(* CODESYS project lclsmotioncontrol.library
   Company: SLAC
   Title: LCLS Motion Control
   Description: A library containing general use motion control POUs for LCLS.
   Placeholder: LCLS Motion Control
   Author: Alex Wallace
   Version: 0.1.2

Project tree, tasks and I/O mapping:
  libraries: LCLS General, * (SLAC); Tc2_MC2, * (Beckhoff Automation GmbH); Tc2_Standard, * (Beckhoff Automation GmbH); Tc2_System, * (Beckhoff Automation GmbH); Tc2_Utilities, * (Beckhoff Automation GmbH); VisuDialogs, * (System)
  POUs/
    GeneralMotion/
      data type E_AxisMotionState
      data type E_AxisMoveMode
      function block FB_BasicAxisControl [ST]: ActError, ActMove, ActPower
      data type ST_BasicAxis
  Version/
    global variables Global_Version
  VISUs/
    visualisation Basic_Axis_PTP
  visualisation Basic_Axis_PTP
  image pool MotionImagePool
  00000000-0000-0000-0000-000000000000|HMI_Images\ccw-icon.svg
  00000000-0000-0000-0000-000000000000|HMI_Images\abs-go-icon.svg
  00000000-0000-0000-0000-000000000000|HMI_Images\rel-cc-icon.svg
  00000000-0000-0000-0000-000000000000|HMI_Images\rel-plus-icon.svg
  00000000-0000-0000-0000-000000000000|HMI_Images\rel-minus-icon.svg
  00000000-0000-0000-0000-000000000000|HMI_Images\stop-icon.svg
*)

// POUs/GeneralMotion/E_AxisMotionState
TYPE E_AxisMotionState :
(
	Init := 10,
	MoveEnabled := 3000,
	Error := 9000
);
END_TYPE

// POUs/GeneralMotion/E_AxisMoveMode
TYPE E_AxisMoveMode :
(
	Hold := 0,
	MoveAbs	:= 1,
	MoveRel	:= 2
) WORD;
END_TYPE

// POUs/GeneralMotion/ST_BasicAxis
TYPE ST_BasicAxis :
STRUCT

(* Controls *)
xEnable	:	BOOL;
rReqAbsPos	:	LREAL;
rReqRelPos	:	LREAL;
xStartRelMovePlus	:	BOOL;
xStartRelMoveMinus	:	BOOL;
xStartAbsMove	:	BOOL;
xStop	:	BOOL;
wMode	:	E_AxisMoveMode;
xReset	:	BOOL;
i_xMotorInterlock	:	BOOL := FALSE; //External motor interlock, overrides axis enable
	
(* Axis motor *)
stAxis	:	AXIS_REF;
lrVelocity	:	LREAL	:=1; //mm/s

eState	:	E_AxisMotionState;

xHiLS	AT %I* :	BOOL;
xLoLS	AT %I* :	BOOL;

END_STRUCT
END_TYPE

// Version/Global_Version
{attribute 'TcGenerated'}
// This function has been automatically generated from the project information.
VAR_GLOBAL CONSTANT
	{attribute 'const_non_replaced'}
	{attribute 'linkalways'}
	stLibVersion_LCLS_Motion_Control : ST_LibVersion := (iMajor := 0, iMinor := 1, iBuild := 2, iRevision := 0, sVersion := '0.1.2');
END_VAR

// POUs/GeneralMotion/FB_BasicAxisControl
FUNCTION_BLOCK FB_BasicAxisControl
VAR_INPUT
END_VAR
VAR_OUTPUT
	q_asResult: ARRAY [1..20] OF STRING;
	q_xError	:	BOOL;
	q_MoveDone	:	BOOL;
END_VAR
VAR_IN_OUT
	iq_Axis	:	ST_BasicAxis;
END_VAR
VAR
	

	mcPower	:	MC_Power;
	mcReset	:	MC_Reset;
	mcMoveAbsolute : MC_MoveAbsolute;
	mcMoveRelative : MC_MoveRelative;
	mcHalt	:	MC_Halt;
	
	//Error Stuff
	indexResult: FB_Index := (LowerLimit:= 1, UpperLimit:=20);
	fbFormatString	:	FB_FormatString;
	
	imcBlockIndex: INT;
	imcBlockIndexPrev : INT;
	
	rtEnable : R_TRIG;
	ftEnable : F_TRIG;
	rtStop	:	R_TRIG;
	rtStartAbsMove	:	R_TRIG;
	rtStartRelMove	:	R_TRIG;
	rReqAbsPosOld: REAL := 0;
	Direction: LREAL := 1;
	i_xMotorInterlock: INT;
	
END_VAR

(* Basic Axis Controls
Alex Wallace, 2016-8-8 

This FB provides limit switch monitoring, and a basic state machine for absolute and relative moves.

We needed a basic control block that would give us some of the functionality of the system manager screen
that is used for commissioning axes.

*)


rtEnable(CLK:=iq_Axis.xEnable);

//Update status
iq_Axis.stAxis();

//Motor Interlock
////////////////////////////////////////////
//If we attempt to enable the motor, but there is an interlock preventing us, log it
IF rtEnable.Q AND NOT iq_Axis.i_xMotorInterlock THEN
	q_asResult[indexResult.IncVal()] := 'Axis enable failed, motor interlock is not satisfied';
END_IF

iq_Axis.xEnable R= NOT iq_Axis.i_xMotorInterlock;
mcPower.Enable := iq_Axis.xEnable AND iq_Axis.i_xMotorInterlock;

ftEnable(CLK:=iq_Axis.xEnable);
//Reset the axis if it is "turned off"/ disabled
IF ftEnable.Q THEN iq_Axis.eState := Init; END_IF

CASE iq_Axis.eState OF
	0: iq_Axis.eState := Init;
	Init:
		(* Start by initializing the motor axis *)
		IF mcPower.Status AND NOT ftEnable.Q THEN //success
			q_asResult[indexResult.IncVal()] := 'Motor init success';
			iq_Axis.eState := MoveEnabled;
		ELSIF mcPower.Error THEN
			mcPower.Enable := FALSE;
			fbFormatString.sFormat:='Init mcPower Error: %#X';
			fbFormatString.arg1:=F_UDINT(mcPower.ErrorID);
			ActError();
		END_IF
		
	MoveEnabled:
		//MoveAbs
		///////////////////////////////////////////////////////
			mcMoveAbsolute.Execute S= iq_Axis.xStartAbsMove AND NOT mcMoveRelative.Busy;
			mcMoveAbsolute.Position := iq_Axis.rReqAbsPos;
			IF mcMoveAbsolute.Done OR 
				mcMoveAbsolute.CommandAborted OR 
				mcMoveAbsolute.Busy THEN
				mcMoveAbsolute.Execute := FALSE;
			ELSIF mcMoveAbsolute.Error THEN
				mcMoveAbsolute.Execute := FALSE;
				fbFormatString.sFormat:='MoveAbsoluteError: %#X'; 
				fbFormatString.arg1:=F_UDINT(mcMoveAbsolute.ErrorID);
				ActError();
			END_IF
		//MoveRel
		//////////////////////////////////////////////////////////////////
			mcMoveRelative.Execute S= (iq_Axis.xStartRelMovePlus OR iq_Axis.xStartRelMoveMinus) AND NOT mcMoveAbsolute.Busy;
			IF iq_Axis.xStartRelMoveMinus THEN Direction := -1; ELSE Direction := 1; END_IF
			mcMoveRelative.Distance := Direction * iq_Axis.rReqRelPos;
			IF mcMoveRelative.Done OR 
				mcMoveRelative.CommandAborted OR 
				mcMoveRelative.Busy THEN 
				mcMoveRelative.Execute := FALSE;
			ELSIF mcMoveRelative.Error THEN
				mcMoveRelative.Execute := FALSE;
				fbFormatString.sFormat:='MoveRelativeError: %#X'; 
				fbFormatString.arg1:=F_UDINT(mcMoveRelative.ErrorID);
				ActError();
			END_IF

		iq_Axis.xStartAbsMove := FALSE;
		iq_Axis.xStartRelMovePlus := FALSE;
		iq_Axis.xStartRelMoveMinus := FALSE;
		//Halt
		mcMoveAbsolute.Execute R= iq_Axis.xStop;
		mcMoveRelative.Execute R= iq_Axis.xStop;
		mcHalt.Execute S= iq_Axis.xStop;
		mcHalt.Execute R= mcHalt.Busy;
		

	Error:
		IF mcReset.Done THEN
			q_xError := FALSE;
			iq_Axis.eState:=Init;
		END_IF
	
END_CASE

//Move done output logic
//Dones aren't reset until the logic block runs again
q_MoveDone := mcMoveRelative.Done OR mcMoveAbsolute.Done;

(* Run the mc blocks *)
ActPower();
iq_Axis.xReset R= mcReset.Done;
mcReset.Execute := iq_Axis.xReset;
mcReset(Axis:=iq_Axis.stAxis);

mcHalt(Axis:=iq_Axis.stAxis);
ActMove();

ACTION ActError:
(* Error action
*)

//Reset the debugging index
iq_Axis.eState := Error;
q_xError	:=	TRUE;
fbFormatString(sOut=>q_asResult[indexResult.IncVal()]);
END_ACTION

ACTION ActMove:
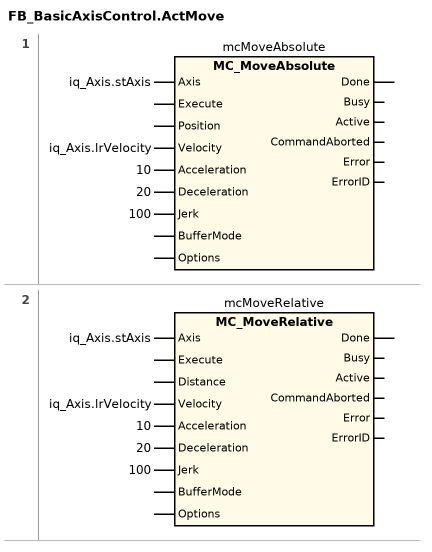
// NETWORK 1
mcMoveAbsolute(
    Axis := iq_Axis.stAxis,
    Velocity := iq_Axis.lrVelocity,
    Acceleration := 10,
    Deceleration := 20,
    Jerk := 100); // MC_MoveAbsolute

// NETWORK 2
mcMoveRelative(
    Axis := iq_Axis.stAxis,
    Velocity := iq_Axis.lrVelocity,
    Acceleration := 10,
    Deceleration := 20,
    Jerk := 100); // MC_MoveRelative
END_ACTION

ACTION ActPower:
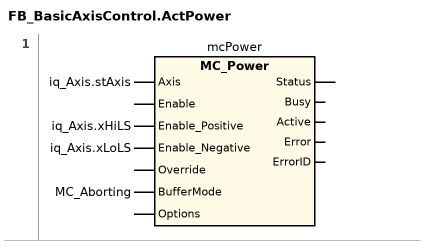
// NETWORK 1
mcPower(
    Axis := iq_Axis.stAxis,
    Enable_Positive := iq_Axis.xHiLS,
    Enable_Negative := iq_Axis.xLoLS,
    BufferMode := MC_Aborting); // MC_Power
END_ACTION

END_FUNCTION_BLOCK

// VISUs/Basic_Axis_PTP
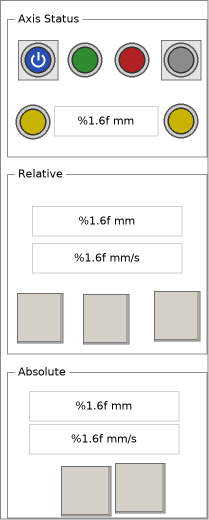
VISUALIZATION Basic_Axis_PTP  // 209x520
VAR_IN_OUT
	stBasicAxis	:	ST_BasicAxis;
END_VAR
    GroupBox (7,11 200x146), "Axis Status"
        PowerSwitch (11,29 40x40), tooltip "Enable Axis", variable: stBasicAxis.xEnable, behaviour: TOGGLE, style: Switch-PowerSwitch-Blue
        Lamp1 (6,91 40x40), tooltip "Minus limit switch is hit", variable: NOT stBasicAxis.xLoLS, style: Lamp-Lamp1-Yellow
        Lamp1 (58,29 40x40), tooltip "Axis enabled", variable: stBasicAxis.stAxis.Status.StandStill OR stBasicAxis.stAxis.Status.Moving, style: Lamp-Lamp1-Green
        Lamp1 (154,90 40x40), tooltip "Plus limit switch is hit", variable: NOT stBasicAxis.xHiLS, style: Lamp-Lamp1-Yellow
        Lamp1 (105,29 40x40), tooltip "Error", variable: stBasicAxis.eState = 9000, style: Lamp-Lamp1-Red
        PushSwitch (154,29 40x40), tooltip "Reset error.", variable: stBasicAxis.xReset, behaviour: TOGGLE, style: Switch-PushSwitch-Gray
        Textfield (47,95 104x30), "%1.6f mm", tooltip "Absolute position", text variable: stBasicAxis.stAxis.NcToPlc.ActPos
    GroupBox (7,364 200x154), "Absolute"
        Button (54,102 50x50), image: MotionImagePool.stop-icon
            tap stBasicAxis.xStop
        Button (108,99 50x50), image: MotionImagePool.rel-plus-icon
            tap stBasicAxis.xStartAbsMove
            OnMouseClick: write the text variable via Default
        Textfield (22,60 150x30), "%1.6f mm/s", text variable: stBasicAxis.lrVelocity
            OnMouseClick: write the text variable via Default
        Textfield (22,27 150x30), "%1.6f mm", text variable: stBasicAxis.rReqAbsPos
            OnMouseDown: write the text variable via Default
    GroupBox (7,166 200x188), "Relative"
        Textfield (25,40 150x30), "%1.6f mm", text variable: stBasicAxis.rReqRelPos
            OnMouseDown: write the text variable via Edit
        Textfield (25,77 150x30), "%1.6f mm/s", text variable: stBasicAxis.lrVelocity
        Button (147,125 46x50), image: MotionImagePool.rel-plus-icon
            tap stBasicAxis.xStartRelMovePlus
        Button (76,128 46x50), image: MotionImagePool.stop-icon
            tap stBasicAxis.xStop
        Button (10,127 46x50), image: MotionImagePool.rel-minus-icon
            tap stBasicAxis.xStartRelMoveMinus
END_VISUALIZATION

// /Basic_Axis_PTP
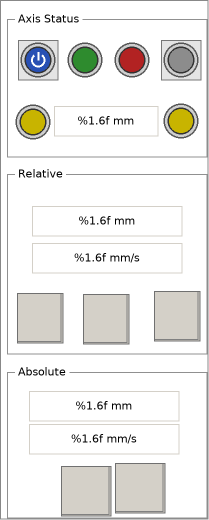
VISUALIZATION Basic_Axis_PTP  // 209x520
VAR_IN_OUT
	stBasicAxis	:	ST_BasicAxis;
END_VAR
    GroupBox (7,11 200x146), "Axis Status"
        PowerSwitch (11,29 40x40), tooltip "Enable Axis", variable: stBasicAxis.xEnable, behaviour: TOGGLE, style: Switch-PowerSwitch-Blue
        Lamp1 (6,91 40x40), tooltip "Minus limit switch is hit", variable: NOT stBasicAxis.xLoLS, style: Lamp-Lamp1-Yellow
        Lamp1 (58,29 40x40), tooltip "Axis enabled", variable: stBasicAxis.stAxis.Status.StandStill OR stBasicAxis.stAxis.Status.Moving, style: Lamp-Lamp1-Green
        Lamp1 (154,90 40x40), tooltip "Plus limit switch is hit", variable: NOT stBasicAxis.xHiLS, style: Lamp-Lamp1-Yellow
        Lamp1 (105,29 40x40), tooltip "Error", variable: stBasicAxis.eState = 9000, style: Lamp-Lamp1-Red
        PushSwitch (154,29 40x40), tooltip "Reset error.", variable: stBasicAxis.xReset, behaviour: TOGGLE, style: Switch-PushSwitch-Gray
        Textfield (47,95 104x30), "%1.6f mm", tooltip "Absolute position", text variable: stBasicAxis.stAxis.NcToPlc.ActPos
    GroupBox (7,364 200x154), "Absolute"
        Button (54,102 50x50), image: MotionImagePool.stop-icon
            tap stBasicAxis.xStop
        Button (108,99 50x50), image: MotionImagePool.rel-plus-icon
            tap stBasicAxis.xStartAbsMove
            OnMouseClick: write the text variable via Default
        Textfield (22,60 150x30), "%1.6f mm/s", text variable: stBasicAxis.lrVelocity
            OnMouseClick: write the text variable via Default
        Textfield (22,27 150x30), "%1.6f mm", text variable: stBasicAxis.rReqAbsPos
            OnMouseDown: write the text variable via Default
    GroupBox (7,166 200x188), "Relative"
        Textfield (25,40 150x30), "%1.6f mm", text variable: stBasicAxis.rReqRelPos
            OnMouseDown: write the text variable via Edit
        Textfield (25,77 150x30), "%1.6f mm/s", text variable: stBasicAxis.lrVelocity
        Button (147,125 46x50), image: MotionImagePool.rel-plus-icon
            tap stBasicAxis.xStartRelMovePlus
        Button (76,128 46x50), image: MotionImagePool.stop-icon
            tap stBasicAxis.xStop
        Button (10,127 46x50), image: MotionImagePool.rel-minus-icon
            tap stBasicAxis.xStartRelMoveMinus
END_VISUALIZATION
